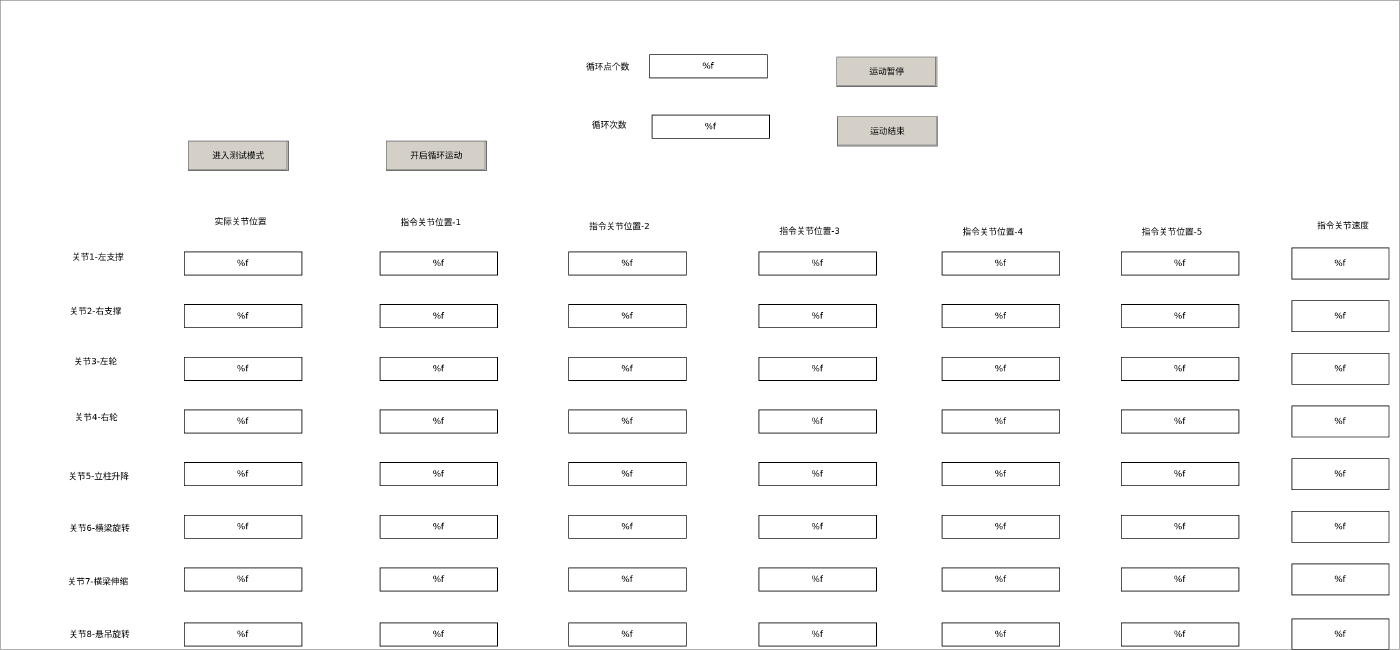
VISUALIZATION cycle_car  // 1781x827
    Label (231,267 150x30), "实际关节位置"
    Rectangle (234,320 150x30), "%f", text variable: g_cycleTest.m_actJntPosCar[1]
    Label (473,268 150x30), "指令关节位置-1"
    Button (239,179 128x38), "进入测试模式", colour toggle: g_cycleTest.m_carEnterCycleTest
        toggle g_cycleTest.m_carEnterCycleTest
    Button (491,179 128x38), "开启循环运动", colour toggle: g_cycleTest.m_startMotionCar
        toggle g_cycleTest.m_startMotionCar
    Rectangle (234,387 150x30), "%f", text variable: g_cycleTest.m_actJntPosCar[2]
    Rectangle (234,454 150x30), "%f", text variable: g_cycleTest.m_actJntPosCar[3]
    Rectangle (234,521 150x30), "%f", text variable: g_cycleTest.m_actJntPosCar[4]
    Rectangle (483,320 150x30), "%f", text variable: g_cycleTest.m_targetJntPosCar[1][1]
        OnMouseClick: write the text variable via Default
    Rectangle (483,387 150x30), "%f", text variable: g_cycleTest.m_targetJntPosCar[1][2]
        OnMouseClick: write the text variable via Default
    Rectangle (483,454 150x30), "%f", text variable: g_cycleTest.m_targetJntPosCar[1][3]
        OnMouseClick: write the text variable via Default
    Rectangle (483,521 150x30), "%f", text variable: g_cycleTest.m_targetJntPosCar[1][4]
        OnMouseClick: write the text variable via Default
    Label (713,273 150x30), "指令关节位置-2"
    Rectangle (723,320 150x30), "%f", text variable: g_cycleTest.m_targetJntPosCar[2][1]
        OnMouseClick: write the text variable via Default
    Rectangle (723,387 150x30), "%f", text variable: g_cycleTest.m_targetJntPosCar[2][2]
        OnMouseClick: write the text variable via Default
    Rectangle (723,454 150x30), "%f", text variable: g_cycleTest.m_targetJntPosCar[2][3]
        OnMouseClick: write the text variable via Default
    Rectangle (723,521 150x30), "%f", text variable: g_cycleTest.m_targetJntPosCar[2][4]
        OnMouseClick: write the text variable via Default
    Label (955,279 150x30), "指令关节位置-3"
    Rectangle (965,320 150x30), "%f", text variable: g_cycleTest.m_targetJntPosCar[3][1]
        OnMouseClick: write the text variable via Default
    Rectangle (965,387 150x30), "%f", text variable: g_cycleTest.m_targetJntPosCar[3][2]
        OnMouseClick: write the text variable via Default
    Rectangle (965,454 150x30), "%f", text variable: g_cycleTest.m_targetJntPosCar[3][3]
        OnMouseClick: write the text variable via Default
    Rectangle (965,521 150x30), "%f", text variable: g_cycleTest.m_targetJntPosCar[3][4]
        OnMouseClick: write the text variable via Default
    Label (1188,280 150x30), "指令关节位置-4"
    Rectangle (1198,320 150x30), "%f", text variable: g_cycleTest.m_targetJntPosCar[4][1]
        OnMouseClick: write the text variable via Default
    Rectangle (1198,387 150x30), "%f", text variable: g_cycleTest.m_targetJntPosCar[4][2]
        OnMouseClick: write the text variable via Default
    Rectangle (1198,454 150x30), "%f", text variable: g_cycleTest.m_targetJntPosCar[4][3]
        OnMouseClick: write the text variable via Default
    Rectangle (1198,521 150x30), "%f", text variable: g_cycleTest.m_targetJntPosCar[4][4]
        OnMouseClick: write the text variable via Default
    Label (1416,280 150x30), "指令关节位置-5"
    Rectangle (1426,320 150x30), "%f", text variable: g_cycleTest.m_targetJntPosCar[5][1]
        OnMouseClick: write the text variable via Default
    Rectangle (1426,387 150x30), "%f", text variable: g_cycleTest.m_targetJntPosCar[5][2]
        OnMouseClick: write the text variable via Default
    Rectangle (1426,454 150x30), "%f", text variable: g_cycleTest.m_targetJntPosCar[5][3]
        OnMouseClick: write the text variable via Default
    Rectangle (1426,521 150x30), "%f", text variable: g_cycleTest.m_targetJntPosCar[5][4]
        OnMouseClick: write the text variable via Default
    Label (698,70 150x30), "循环点个数"
    Rectangle (826,69 150x30), "%f", text variable: g_cycleTest.m_pointSumCar
        OnMouseClick: write the text variable via Default
    Rectangle (829,146 150x30), "%f", text variable: g_cycleTest.m_targetCycleNumCar
        OnMouseClick: write the text variable via Default
    Label (700,144 150x30), "循环次数"
    Button (1064,72 128x38), "运动暂停", colour toggle: g_cycleTest.m_pauseCar
        toggle g_cycleTest.m_pauseCar
    Button (1065,148 128x38), "运动结束", colour toggle: g_cycleTest.m_finishCar
        tap g_cycleTest.m_finishCar
    Rectangle (234,588 150x30), "%f", text variable: g_cycleTest.m_actJntPosCar[5]
    Rectangle (234,655 150x30), "%f", text variable: g_cycleTest.m_actJntPosCar[6]
    Rectangle (234,722 150x30), "%f", text variable: g_cycleTest.m_actJntPosCar[7]
    Rectangle (234,792 150x30), "%f", text variable: g_cycleTest.m_actJntPosCar[8]
    Rectangle (483,588 150x30), "%f", text variable: g_cycleTest.m_targetJntPosCar[1][5]
        OnMouseClick: write the text variable via Default
    Rectangle (483,655 150x30), "%f", text variable: g_cycleTest.m_targetJntPosCar[1][6]
        OnMouseClick: write the text variable via Default
    Rectangle (483,722 150x30), "%f", text variable: g_cycleTest.m_targetJntPosCar[1][7]
        OnMouseClick: write the text variable via Default
    Rectangle (483,792 150x30), "%f", text variable: g_cycleTest.m_targetJntPosCar[1][8]
        OnMouseClick: write the text variable via Default
    Rectangle (723,588 150x30), "%f", text variable: g_cycleTest.m_targetJntPosCar[2][5]
        OnMouseClick: write the text variable via Default
    Rectangle (723,655 150x30), "%f", text variable: g_cycleTest.m_targetJntPosCar[2][6]
        OnMouseClick: write the text variable via Default
    Rectangle (723,722 150x30), "%f", text variable: g_cycleTest.m_targetJntPosCar[2][7]
        OnMouseClick: write the text variable via Default
    Rectangle (723,792 150x30), "%f", text variable: g_cycleTest.m_targetJntPosCar[2][8]
        OnMouseClick: write the text variable via Default
    Rectangle (965,588 150x30), "%f", text variable: g_cycleTest.m_targetJntPosCar[3][5]
        OnMouseClick: write the text variable via Default
    Rectangle (965,655 150x30), "%f", text variable: g_cycleTest.m_targetJntPosCar[3][6]
        OnMouseClick: write the text variable via Default
    Rectangle (965,722 150x30), "%f", text variable: g_cycleTest.m_targetJntPosCar[3][7]
        OnMouseClick: write the text variable via Default
    Rectangle (965,792 150x30), "%f", text variable: g_cycleTest.m_targetJntPosCar[3][8]
        OnMouseClick: write the text variable via Default
    Rectangle (1198,588 150x30), "%f", text variable: g_cycleTest.m_targetJntPosCar[4][5]
        OnMouseClick: write the text variable via Default
    Rectangle (1198,655 150x30), "%f", text variable: g_cycleTest.m_targetJntPosCar[4][6]
        OnMouseClick: write the text variable via Default
    Rectangle (1198,722 150x30), "%f", text variable: g_cycleTest.m_targetJntPosCar[4][7]
        OnMouseClick: write the text variable via Default
    Rectangle (1198,792 150x30), "%f", text variable: g_cycleTest.m_targetJntPosCar[4][8]
        OnMouseClick: write the text variable via Default
    Rectangle (1426,588 150x30), "%f", text variable: g_cycleTest.m_targetJntPosCar[5][5]
        OnMouseClick: write the text variable via Default
    Rectangle (1426,655 150x30), "%f", text variable: g_cycleTest.m_targetJntPosCar[5][6]
        OnMouseClick: write the text variable via Default
    Rectangle (1426,722 150x30), "%f", text variable: g_cycleTest.m_targetJntPosCar[5][7]
        OnMouseClick: write the text variable via Default
    Rectangle (1426,792 150x30), "%f", text variable: g_cycleTest.m_targetJntPosCar[5][8]
        OnMouseClick: write the text variable via Default
    Label (1636,273 145x28), "指令关节速度"
    Rectangle (1643,315 124x40), "%f", text variable: g_cycleTest.m_targetJntVelCar[1]
        OnMouseClick: write the text variable via Default
    Rectangle (1643,382 124x40), "%f", text variable: g_cycleTest.m_targetJntVelCar[2]
        OnMouseClick: write the text variable via Default
    Rectangle (1643,449 124x40), "%f", text variable: g_cycleTest.m_targetJntVelCar[3]
        OnMouseClick: write the text variable via Default
    Rectangle (1643,516 124x40), "%f", text variable: g_cycleTest.m_targetJntVelCar[4]
        OnMouseClick: write the text variable via Default
    Rectangle (1643,583 124x40), "%f", text variable: g_cycleTest.m_targetJntVelCar[5]
        OnMouseClick: write the text variable via Default
    Rectangle (1643,650 124x40), "%f", text variable: g_cycleTest.m_targetJntVelCar[6]
        OnMouseClick: write the text variable via Default
    Rectangle (1643,717 124x40), "%f", text variable: g_cycleTest.m_targetJntVelCar[7]
        OnMouseClick: write the text variable via Default
    Rectangle (1643,787 124x40), "%f", text variable: g_cycleTest.m_targetJntVelCar[8]
        OnMouseClick: write the text variable via Default
    Label (52,313 145x28), "关节1-左支撑"
    Label (49,382 145x28), "关节2-右支撑"
    Label (49,446 145x28), "关节3-左轮"
    Label (50,517 145x28), "关节4-右轮"
    Label (53,592 145x28), "关节5-立柱升降"
    Label (54,658 145x28), "关节6-横梁旋转"
    Label (52,726 145x28), "关节7-横梁伸缩"
    Label (54,793 145x28), "关节8-悬吊旋转"
END_VISUALIZATION

(* stored: Version 1.1.0.1, ProductVersion 3.1.4024.11
   Visu cycle_car: Id {023e9b0b-9b13-4b15-95cc-2be194297f02} *)
